FUNCTION_BLOCK ADP_IDENTIFICATION (* Offline identification prototype; see docs/adaptive/4diac-design.md *)
  (* Standard: 61499-2 *)
  (* Version 0.1, 2026-09-26, Guilherme *)
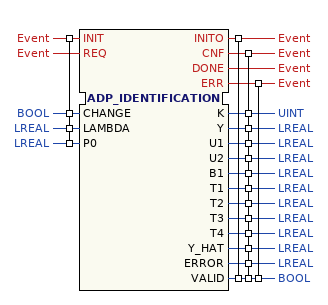
  EVENT_INPUT
    INIT WITH CHANGE, LAMBDA, P0;
    REQ;
  END_EVENT
  EVENT_OUTPUT
    INITO WITH VALID;
    CNF WITH K, Y, U1, U2, B1, T1, T2, T3, T4, Y_HAT, ERROR, VALID;
    DONE;
    ERR WITH VALID;
  END_EVENT
  VAR_INPUT
    CHANGE : BOOL := FALSE;
    LAMBDA : LREAL := 1.0;
    P0 : LREAL := 10000.0;
  END_VAR
  VAR_OUTPUT
    K : UINT;
    Y : LREAL;
    U1 : LREAL;
    U2 : LREAL;
    B1 : LREAL;
    T1 : LREAL;
    T2 : LREAL;
    T3 : LREAL;
    T4 : LREAL;
    Y_HAT : LREAL;
    ERROR : LREAL;
    VALID : BOOL;
  END_VAR
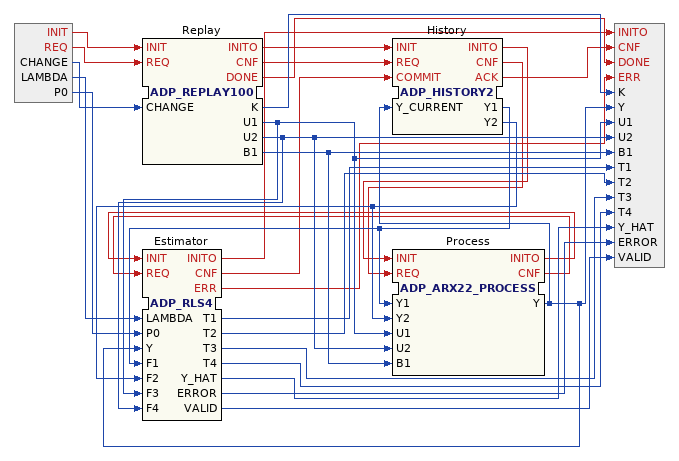
  FBS
    Replay : ADP_REPLAY100;
    History : ADP_HISTORY2;
    Process : ADP_ARX22_PROCESS;
    Estimator : ADP_RLS4;
  END_FBS
  EVENT_CONNECTIONS
    INIT TO Replay.INIT;
    Replay.INITO TO History.INIT;
    History.INITO TO Process.INIT;
    Process.INITO TO Estimator.INIT;
    Estimator.INITO TO INITO;
    REQ TO Replay.REQ;
    Replay.CNF TO History.REQ;
    History.CNF TO Process.REQ;
    Process.CNF TO Estimator.REQ;
    Estimator.CNF TO History.COMMIT;
    History.ACK TO CNF;
    Replay.DONE TO DONE;
    Estimator.ERR TO ERR;
  END_CONNECTIONS
  DATA_CONNECTIONS
    CHANGE TO Replay.CHANGE;
    LAMBDA TO Estimator.LAMBDA;
    P0 TO Estimator.P0;
    Process.Y TO Estimator.Y;
    Process.Y TO History.Y_CURRENT;
    Process.Y TO Y;
    Replay.U1 TO Process.U1;
    Replay.U1 TO U1;
    Replay.U2 TO Process.U2;
    Replay.U2 TO U2;
    Replay.B1 TO Process.B1;
    Replay.B1 TO B1;
    Replay.K TO K;
    History.Y1 TO Process.Y1;
    History.Y1 TO Estimator.F1;
    History.Y2 TO Process.Y2;
    History.Y2 TO Estimator.F2;
    Replay.U1 TO Estimator.F3;
    Replay.U2 TO Estimator.F4;
    Estimator.T1 TO T1;
    Estimator.T2 TO T2;
    Estimator.T3 TO T3;
    Estimator.T4 TO T4;
    Estimator.Y_HAT TO Y_HAT;
    Estimator.ERROR TO ERROR;
    Estimator.VALID TO VALID;
  END_CONNECTIONS
END_FUNCTION_BLOCK
